{attribute 'qualified_only'}
VAR_GLOBAL
	bAutoMode : BOOL; 
	bManualMode : BOOL; 
	fJoyY : LREAL;
END_VAR

(* stored: Version 1.1.0.1, ProductVersion 3.1.4024.10
   GVL Inputs: Id {566405ba-476e-4000-8931-6791d6e2fe7f} *)
